# B&R Automation Studio project TD52 (part 4)

#### UniAna_in.st - Implementation file
```iecst
(********************************************************************
 * COPYRIGHT -- INNIO Company, Zengerer
 ********************************************************************
 * Library: AnalogIn
 * File: AnalogIn.st
 * Author: ZengereS
 * Created: December 04, 2007
 ********************************************************************
 *
 * Description of library AnalogIn:
 ********************************************************************
 *  Function depending on ucInputType:
 *  ---------------------------------
 * 		 0=AI_NO_SCALING: 		(Temperature) Inputs  NO SCALING, NO CLAMPING (PT100 or Thermocouples on ATxx- Units, read in 1/10°C)
 *
 * 	THESE INPUT TYPES ARE CLAMPED: (ssScalMin < ssOut < ssScalMax)
 * 		 1=AI_FixedFactor10:	Temperature inputs (PT100, KTY..... WITH FIXED x10 SCALING TO 1°C; CLAMPED
 *		 2=AI_MA_INPUT:			+-20mA input (-32768 to 32767Digits) scaled to ScalMin-ScalMax; CLAMPED
 *		 3=AI_0-20MA_INPUT:		0-20mA input (0-32767Digits) scaled to ScalMin-ScalMax; CLAMPED
 *		 4=AI_4_20MA_INPUT:		4-20mA input (6554-32767Digits) scaled to ScalMin-ScalMax; CLAMPED
  *		 5=AI_0_5V_INPUT:		0-5V input (0-16364Digits) scaled to ScalMin-ScalMax; CLAMPED		(NEW)
 * 		 9=AI_NO_SCALING, CLAMPED: (Temperature) Inputs  NO SCALING (PT100 or Thermocouples on ATxx- Units, read in 1/10°C) ; CLAMPED BETWEEN ScalMin and ScalMax
 *
 *	THESE INPUT TYPES ARE ALLSO AVAILABLE WITHOUT CLAMPING: (ssScalMin <> ssOut <> ssScalMax)
 * 		11=AI_FixedFactor10:	NO CLAMPING Temperature inputs (PT100, KTY..... WITH FIXED x10 SCALING TO 1°C (usage not recommendet)
 *		12=AI_MA_INPUT:			NO CLAMPING +-20mA input (-32768 to 32767Digits) scaled to ScalMin-ScalMax    (usage not recommendet))
 *		13=AI_0-20MA_INPUT:		NO CLAMPING 0-20mA input (0-32767Digits) scaled to ScalMin-ScalMax
 *		14=AI_4_20MA_INPUT:		NO CLAMPING 4-20mA input (6554-32767Digits) scaled to ScalMin-ScalMax
 *		15=AI_0_5V_INPUT:		0-5V input (0-16364Digits) scaled to ScalMin-ScalMax
 *
 *	!scNrOfDecimal WORKS AS MULTIPLIER FOR THE SCALED VALUE BY SHIFTING THE DECIMAL POINT!
 *
 *	DEFINE OUTPUT CHANNELS WITH THESE TYPE CODES: (same sScalMin and ssScalMax are applied to Output signal) (NEESDS EXTERNAL CODE PARTS!)
 * 		11=AI_0-20MA_INPUT:		0-20mA output (0-32767Digits) scaled from channel signal ScalMin-ScalMax (input behavior typ 0, if HW input stays connected!)
 *		24=AI_4_20MA_OUTPUT:	4-20mA output (6554-32767Digits) scaled from channel signal ScalMin-ScalMax (input behavior typ 0, if HW in connected!)
 *
 *
 *  SPECIAL CODES FOR 'usANDLinkNum' (Numbers 1 to 250 are reserved for the channel numbers to add another channel value)
 *		 253=RawManualValue:		Enter MANUAL RAW VALUE in ssManualValue for overriding input
 *		 254=AddManualValue:		Enter MANUAL ADD VALUE in ssManualValue as addition summand to the scaled output
 *		 255=UseManualValue:		Enter MANUAL OVERRIDE VALUE in ssManualValue for direct output
 *
 *	Limit activation with ucOtionBits:
 *  	bErrOptiMin	:= activation with ucOptionBits = 1
 *		bErrOptiMax := activation with ucOptionBits = 2
 *		bErrMin		:= activation with ucOptionBits = 4
 *		bErrMax		:= activation with ucOptionBits = 8
 *		bErrMINMIN	:= activation with ucOptionBits = 16
 *		bErrMAXMAX	:= activation with ucOptionBits = 32

 *  	bErrSignal	:= DEactivation with ucOptionBits = 64   (MEASUREMENT SIGNAL DETECTION-> ALARM)
 *
 ********************************************************************
 *  History:
 *  --------
 *	2008-09-10  V0.20	Zengerer	added scaling calculations
 *	2008-09-11  V0.21	Zengerer	added Helper Structure for old SG3- visu
 *	2008-09-30  V0.22	Zengerer	added texts and color changing
 *	2008-09-30  V0.23	Zengerer	added Input Types 10-14 for unclamped values wihout limitation between Min/Max scaling
 *	2008-10-22  V0.30	Zengerer	CHANGED CONFIGTYPE: scNrOfDecimal instead of ucNrOfDecimal
 *	2009-05-22	V0.40	Zengerer	Limit activation with OtionBits masking
 *	2009-06-22	V0.42	Zengerer	Limit OptionBits update
 *  2010-06-04  V0.50	Zengerer	NAMETEXT expanded to 32 CHARACTERS; ssManualValue and usANDLinkNum new introduced in datatype
  *	2009-11-25	V0.50	Zengerer	0-5V Inputtype added
 *	2010-06-22	V0.51	Zengerer	predefined system value in 'usANDLinkNum' removed here, externaly realised
 *	2010-06-22	V0.52	Zengerer	additional infotext for output types (output handling externaly realised)
 *	2010-06-22	V0.60	Zengerer	Manual override of RAW value! with linkCode 253
 *	2013-10-31	V0.70	Zengerer	FILTER type as local implemented function to cancel dependency on JEW_LIB1
 *  2013-11-11  V0.71	Zengerer	Filter function reverted-  has to stay in task
*
* LEGACY CODE- DO NOT USE IN NEW IMPLEMENTATIONS!
*
 ********************************************************************)

FUNCTION_BLOCK ana_in		(*Analogeingang oder Temperatureingang*)

	IF tAnaInPERMEM.bEnable THEN					(*1=enable input*)
		(*get InputType from parameterstructure: types 1-9 are clamped to min/max EU, types 11-19 are proceedet like 1-9, but without clamping*)
		IF tAnaInPERMEM.ucInputType >9 AND tAnaInPERMEM.ucInputType <19 THEN
			ucInputType	:= tAnaInPERMEM.ucInputType -10;					(*Internal use: input type only from 0-8*)
		ELSE
			ucInputType	:= tAnaInPERMEM.ucInputType ;						(*Internal use: input type only from 0-8*)
			IF tAnaInPERMEM.ucInputType = 9 THEN ucInputType := 0; END_IF	(*Internal use: input type only from 0-8*)
		END_IF

		(*Statustext output*)
		CASE ucInputType OF
			0:		(*AI_NO_SCALING '1234567890123456'*)
					szOutState	:= 	'UnscaledIn(Temp)';
	 		1:		(*AI_AI_FixedFactor10     *)
					szOutState	:= 	'Temp.Input X°C';
			2:		(*AI_-10+10V_INPUT*)
					szOutState	:= 	'+-10V Input OK';
			3:		(*AI_0-20MA_INPUT*)
					szOutState	:= 	'0-20mA OK';
			4:		(*AI_4_20MA_INPUT*)
					szOutState	:= 	'4-20mA OK';
			5:		(*AI_0_5V_INPUT*)
					szOutState	:= 	'+5V Input';
			9:		(*AI_NO_SCALING '1234567890123456'*)
					szOutState	:= 	'Unscaled Clamped';
	 		11:		(*AI_AI_FixedFactor10     *)
					szOutState	:= 	'Temp.Inp.NoClamp';
			12:		(*AI_-10+10V_INPUT*)
					szOutState	:= 	'+-10V In.NoClamp';
			13:		(*AI_0-20MA_INPUT*)
					szOutState	:= 	'0-20mA NoClamp';
			14:		(*AI_4_20MA_INPUT*)
					szOutState	:= 	'4-20mA NoClamp';
			15:		(*AI_0_5V_INPUT*)
					szOutState	:= 	'+5V Inp. NoClamp';
			23:		(*AI_0-20MA_OUTPUT*)
					szOutState	:= 	'0-20mA OUTPUT OK';
			24:		(*AI_4-20MA_OUTPUT*)
					szOutState	:= 	'4-20mA OUTPUT OK';
		ELSE		(*CASE_ELSE*)
					szOutState	:= 	'NoTypeInfo';
		END_CASE

		(*Manual override of RAW value! with linkCode 253 (watch external code allso!*)
		IF tAnaInPERMEM.usANDLinkNum =253 THEN
			ssIn := tAnaInPERMEM.ssManualValue;
		 	szOutState	:= 	'MANUAL RAW VALUE';
		END_IF

		(*SIGNAL FAILURE DETECTION*)
		CASE ucInputType OF
			0:		(*AI_NO_SCALING:  (Temperature inputs PT100, Termocouples == 1/10°C from ATxx Units WITHOUT SCALING *)
				tAna_inErrors.bErrSignal := (ssIn < LIM_PT100_MIN OR ssIn > LIM_PT100_MAX);
			1:		(*AI_AI_FixedFactor10:  (temperature) inputs WITH x10 SCALING to convert to 1°C*)
				tAna_inErrors.bErrSignal := ((ssIn/10) < LIM_PT100_MIN OR (ssIn/10) > LIM_PT100_MAX);
		    2:		(*AI_-10+10V_INPUT*)
				tAna_inErrors.bErrSignal := FALSE;   (*NO SIGNAL CHECK!*)  (* (ssIn < LIM_MA_MIN) *OR ssIn > LIM_MA_MAX); *)
			3:		(*AI_0_20MA_INPUT*)
				tAna_inErrors.bErrSignal := (ssIn < LIM_0_20MA_MIN); (*OR ssIn > LIM_0_20MA_MAX);*)
			4:		(*AI_4_20MA_INPUT*)
				tAna_inErrors.bErrSignal := (ssIn < LIM_4_20MA_MIN); (*OR ssIn > LIM_4_20MA_MAX);*)
			5:		(*AI_0_5V_INPUT*)
				tAna_inErrors.bErrSignal := (ssIn < LIM_0_5V_MIN OR ssIn > LIM_0_5V_MAX);
			9:		(*AI_NO_SCALING, clamped*)
				tAna_inErrors.bErrSignal := (ssIn < LIM_PT100_MIN OR ssIn > LIM_PT100_MAX);
		ELSE		(*CASE_ELSE*)
				tAna_inErrors.bErrSignal := FALSE;

		END_CASE

		(*INPUT SIGNAL FILTER*)
		FILTER_0(In := ssIn, Filter := UINT_TO_USINT(tAnaInPERMEM.usSetFilterValue) );			(*FILTER type local implementedr function to cancel dependency on JEW_LIB1 *)

		IF tAna_inErrors.bErrSignal  THEN
			ssInFiltered := DINT_TO_INT(FILTER_0.Out);
		ELSE
			ssInFiltered := ssIn;		(*unfiltered, to shorten reaction time on signal newstart *)
		END_IF

		(*INPUT SCALING*)
		CASE ucInputType OF
			0:		(*AI_PT100_NO_SCALING*)
					slOutScaled		:= 	INT_TO_DINT( ssInFiltered );
	 		1:		(*AI_AI_FixedFactor10*)
					slOutScaled		:= 	INT_TO_DINT( ssInFiltered ) / 10 ;
			2:		(*AI_-10+10V_INPUT*)
					slOutScaled		:=  (INT_TO_DINT(ssInFiltered) + 32768 ) * (tAnaInPERMEM.ssScalMax - tAnaInPERMEM.ssScalMin) / (32767*2) + tAnaInPERMEM.ssScalMin ;
			3:		(*AI_0-20MA_INPUT*)
					slOutScaled		:= 	(INT_TO_DINT(ssInFiltered)         ) * (tAnaInPERMEM.ssScalMax - tAnaInPERMEM.ssScalMin) / 32768 + tAnaInPERMEM.ssScalMin ;
			4:		(*AI_4_20MA_INPUT*)
					slOutScaled		:=  (INT_TO_DINT(ssInFiltered) - 6554  ) * (tAnaInPERMEM.ssScalMax - tAnaInPERMEM.ssScalMin) / (32768-6554) + tAnaInPERMEM.ssScalMin ;
			5:		(*AI_0_5V_INPUT*)
					slOutScaled		:= 	(INT_TO_DINT(ssInFiltered)         ) * (tAnaInPERMEM.ssScalMax - tAnaInPERMEM.ssScalMin) / 16383 + tAnaInPERMEM.ssScalMin ;			(*scaling 100% = only 50% of electrical max+ to use a +-10V input*)
			9:		(*AI_PT100_NO_SCALING, clamped*)
					slOutScaled		:= 	INT_TO_DINT( ssInFiltered );
		ELSE		(*CASE_ELSE*)
					slOutScaled		:= 	0;
		END_CASE

		(*INPUT CLAMPING on Min-Max scaling parameters*)
		IF tAnaInPERMEM.ucInputType > 0 AND tAnaInPERMEM.ucInputType < 10 THEN	(*all input types with codenumber 1-9 get their output values clamped*)
			IF slOutScaled < tAnaInPERMEM.ssScalMin	THEN slOutScaled := tAnaInPERMEM.ssScalMin;	END_IF
			IF slOutScaled > tAnaInPERMEM.ssScalMax	THEN slOutScaled := tAnaInPERMEM.ssScalMax;	END_IF
		END_IF

		(*OPTION: Calculate combined value of this and another channel*)
		IF tAnaInPERMEM.usANDLinkNum > 0 AND tAnaInPERMEM.usANDLinkNum < 251 THEN
  			(*tAnaInPERMEM.usANDLinkNum; *)  					  	(*!!!	EXTERN realisiert   !!!*)
		 	szOutState	:= 	'Channel x Val.ad';
		END_IF

		(*Add manual value optional with linkCode 254 *)
		IF tAnaInPERMEM.usANDLinkNum =254 THEN
			slOutScaled := slOutScaled + tAnaInPERMEM.ssManualValue;
		 	szOutState	:= 	'Manualvalue add.';
		END_IF
		(*Manual override! with linkCode 255*)
		IF tAnaInPERMEM.usANDLinkNum =255 THEN
			slOutScaled := tAnaInPERMEM.ssManualValue;
		 	szOutState	:= 	'Manual Override';
		END_IF

		(*INPUT CLAMPING ONCE MORE FOR ADDED VALUES*)
		IF tAnaInPERMEM.ucInputType > 0 AND tAnaInPERMEM.ucInputType < 10 THEN	(*all input types with codenumber 1-9 get their output values clamped*)
			IF slOutScaled < tAnaInPERMEM.ssScalMin	THEN slOutScaled := tAnaInPERMEM.ssScalMin;	END_IF
			IF slOutScaled > tAnaInPERMEM.ssScalMax	THEN slOutScaled := tAnaInPERMEM.ssScalMax;	END_IF
		END_IF

		(*OUTPUT TO INTEGER Variable*)
		ssOut 	:= DINT_TO_INT( slOutScaled );
		IF slOutScaled < -32768		THEN ssOut := -32768;	END_IF		(* (just to be sure...) *)
		IF slOutScaled > 32767		THEN ssOut := 32767; 	END_IF   	(* (just to be sure...) *)

		(*		ssOutMod 	:= MOD(ssInFiltered,10);   ALT *)

		(*LIMITS*)
		(*Limit activation with OtionBits masking:  NOT AND=0 (XOR) *)
			tAna_inErrors.bErrOptiMin	:= 	(NOT( (tAnaInPERMEM.ucOptionBits AND 1) =0) ) 		AND (ssOut < tAnaInPERMEM.ssSetPointOptiMin);
  			tAna_inErrors.bErrMin		:= 	(NOT( (tAnaInPERMEM.ucOptionBits AND 4) =0) )		AND (ssOut < tAnaInPERMEM.ssSetPointMin);
  			tAna_inErrors.bErrMINMIN	:= 	(NOT( (tAnaInPERMEM.ucOptionBits AND 16)=0) )		AND (ssOut < tAnaInPERMEM.ssSetPointMINMIN);
			tAna_inErrors.bErrOptiMax	:= 	(NOT( (tAnaInPERMEM.ucOptionBits AND 2) =0) )		AND (ssOut > tAnaInPERMEM.ssSetPointOptiMax);
			tAna_inErrors.bErrMax		:= 	(NOT( (tAnaInPERMEM.ucOptionBits AND 8) =0) )		AND (ssOut > tAnaInPERMEM.ssSetPointMax);
			tAna_inErrors.bErrMAXMAX	:= 	(NOT( (tAnaInPERMEM.ucOptionBits AND 32)=0) )		AND (ssOut > tAnaInPERMEM.ssSetPointMAXMAX);

			(*Statustext Messages for Limits    				'12345678901234'   *)
			IF tAna_inErrors.bErrOptiMin		THEN szOutState	:= 	'<OptiMin exc. '; 	END_IF
			IF tAna_inErrors.bErrMin 			THEN szOutState	:= 	'<Min Limit    '; 	END_IF
			IF tAna_inErrors.bErrMINMIN 		THEN szOutState	:= 	'<MINMIN Limit!'; 	END_IF
			IF tAna_inErrors.bErrOptiMax		THEN szOutState	:= 	'>OptiMax exc. '; 	END_IF
			IF tAna_inErrors.bErrMax 			THEN szOutState	:= 	'>Max Limit    '; 	END_IF
			IF tAna_inErrors.bErrMAXMAX 		THEN szOutState	:= 	'>MAXMAX Limit!'; 	END_IF

		(*Check limit values valid?*)
		(*	IF 	tAnaInPERMEM.bOptSupervice AND*)
   			IF	(NOT( (tAnaInPERMEM.ucOptionBits AND 8)=1 ))	AND			(*Optionsbit für ErrMINMIN ausmaskieren*)
				(NOT( (tAnaInPERMEM.ucOptionBits AND 64)=1 ))	AND			(*Optionsbit für ErrMAXMAX ausmaskieren*)
   				(tAnaInPERMEM.ssSetPointMINMIN = 0) AND
   				(tAnaInPERMEM.ssSetPointMAXMAX <= tAnaInPERMEM.ssSetPointMINMIN)
			THEN
				tAna_inErrors.bErrMINMIN	:= FALSE;
				tAna_inErrors.bErrMAXMAX	:= FALSE;
				szOutState	:= 	'LimitsNotValid';
			END_IF

		IF tAna_inErrors.bErrSignal  THEN	szOutState	:= 	'OutOfRange'; END_IF

		(*failed signal check sets output to 'errorvalue' *)
		IF tAna_inErrors.bErrSignal AND NOT (tAnaInPERMEM.usANDLinkNum =255) THEN
			ssOut		:= -9999;
(*			ssOutModulo	:= -9999; 	*)
		END_IF
		IF tAnaInPERMEM.usANDLinkNum =255 THEN	szOutState	:= 	'Manual Override!'; 	END_IF 	(*this messagetext has priotity and overrides the one before!*)

		(*Quittierung...*)
			bInQuit;
		(* 	bOutErr		:= FALSE;
		(*FEHLT NOCH!!!*)

		(*Config Mode*)
		(*FEHLT NOCH!!!*)
		(*bConfigModeActive;*)

	ELSE						(* else to .bEnable: 0=disables all input functions*)
		ssOut		:= 0;
		ssOutModulo	:= 0;
		rOut		:= 0;
		tAna_inErrors.bErrSignal 	:= 	FALSE;
		tAna_inErrors.bErrMAXMAX	:= 	FALSE;
		tAna_inErrors.bErrMax		:= 	FALSE;
		tAna_inErrors.bErrOptiMax	:= 	FALSE;
		tAna_inErrors.bErrOptiMin	:= 	FALSE;
		tAna_inErrors.bErrMin		:= 	FALSE;
		tAna_inErrors.bErrMINMIN	:= 	FALSE;
		szOutState	:= 	'DISABELED';

	END_IF

	(*Alternative: output as scaled real value*)
(*OLD	CASE tAnaInPERMEM.scNrOfDecimal  OF
			-1:		(**)
(*					rOut			:= INT_TO_REAL(ssOutScaled) *10 ;
			0:
(*					rOut			:= INT_TO_REAL(ssOutScaled);
			1:		(**)
(*					rOut			:= INT_TO_REAL(ssOutScaled) /10 ;
			2:		(**)
(*					rOut			:= INT_TO_REAL(ssOutScaled) /100 ;
			3:		(**)
(*					rOut			:= INT_TO_REAL(ssOutScaled) /1000 ;
			4:		(**)
(*					rOut			:= INT_TO_REAL(ssOutScaled) /10000 ;
	ELSE		(*CASE_ELSE*)
(*					rOut			:= 0 ;
	END_CASE		(**)

		rOut		:= DINT_TO_REAL(slOutScaled)  * EXPT(10 , -tAnaInPERMEM.scNrOfDecimal) ;  (* ...*10^(-NrOfDecimal) VORSICHT: NICHT IEC1131 -Konform!!*)

END_FUNCTION_BLOCK

(******************************************************************************)
(******************************************************************************)
(******************************************************************************)

FUNCTION_BLOCK ana_in_SG3helper		(*stellt mit Informationen aus ana_in zusäzlichen Statusausgängen für alte SG3- Visu zur Verfügung*)

		(*outputs for local paneldisplay*)
(*OLD*		CASE ucInputType OF
(*	 		0:		(*AI_NO_SCALING*)
(*					ssOutRaw		:= 	DINT_TO_INT( LIMIT( (INT_TO_DINT(ssInRaw)   * 32767  / 2000 )    , 0, 32767) ); (*scale 0-200°C to full display range*)
(*			1:		(*AI_PT100_NO_SCALING*)
(*					ssOutRaw		:= 	DINT_TO_INT( LIMIT( (INT_TO_DINT(ssInRaw)   * 32767  / 2000 )    , 0, 32767) ); (*scale 0-200°C to full display range*)
(*			2:		(*AI_-10+10V_INPUT*)
(*					ssOutRaw		:= 	LIMIT( ABS( ssInRaw )  	, 0, 32767);
(*			3:		(*AI_0-20MA_INPUT*)
(*					ssOutRaw		:= 	LIMIT( ssInRaw  		, 0, 32767);
(*			4:		(*AI_4_20MA_INPUT*)
(*					ssOutRaw		:= 	LIMIT( ssInRaw  		, 0, 32767);
(*		ELSE
(*					ssOutRaw		:= 	LIMIT( ssInRaw  		, 0, 32767);
(*		END_CASE
(*\OLD*)
	(*	ssOutRaw		:= 	REAL_TO_INT( LOG( INT_TO_REAL(ssInRaw) / 100 ) * 13000 );		(*logarythmic bargraph scaling*)
	(*	ssOutRaw		:= 	REAL_TO_INT( LN( INT_TO_REAL(ssInRaw) ) * 3150 );		(*logarythmic bargraph scaling*)
		ssOutRaw		:= 	REAL_TO_INT( SQRT( INT_TO_REAL(ssInRaw) ) * 181 );		(*exponential bargraph scaling*)

		(*OPTIONAL: outputs scaled for local paneldisplay with fixed 3 digits after decimal*)
		CASE tAnaInPERMEM.scNrOfDecimal  OF
	 		0:
					slOut			:= DINT_TO_INT(ssIn) * 1000;
			1:		(**)
					slOut			:= DINT_TO_INT(ssIn) * 100 ;
			2:		(**)
					slOut			:= DINT_TO_INT(ssIn) * 10;
			3:		(**)
					slOut			:= DINT_TO_INT(ssIn) * 1;
			4:		(**)
					slOut			:= DINT_TO_INT(ssIn) / 10;

		ELSE		(*CASE_ELSE*)
					slOut			:= 0 ;
		END_CASE

	(*SG3 VISU: HELPER OUTPUTS to activate displays and change colors*)
 	tAnaInHelper.ucStatus	:= 93;														(* blue and INvisible (set 1-bit == uneven decimal colornumber)*)
	IF  tAnaInPERMEM.bEnable	 THEN
 		tAnaInHelper.ucStatus	:= 10;													(* green and visible (no 1-bit! == only even decimal numbers)*)
		IF 	tAna_inErrors.bErrOptiMax OR tAna_inErrors.bErrOptiMin	THEN  	tAnaInHelper.ucStatus := 142; END_IF	(* (ligth)green and visible (no 1-bit!*)
		IF 	tAna_inErrors.bErrMax OR tAna_inErrors.bErrMin			THEN  	tAnaInHelper.ucStatus := 040; END_IF	(* yellow and visible (no 1-bit!*)
		IF 	tAna_inErrors.bErrMAXMAX OR tAna_inErrors.bErrMINMIN	THEN  	tAnaInHelper.ucStatus := 050; END_IF	(* red and visible (no 1-bit!*)
  		IF 	tAna_inErrors.bErrSignal								THEN  	tAnaInHelper.ucStatus := 038; END_IF	(* red and visible (no 1-bit!*)
		IF ssInRaw < - 4											THEN	tAnaInHelper.ucStatus := 246; END_IF	(* NEGATIVE RAW VALUES showed liggthblue and visible (no 1-bit!*)

	(*SG3 VISU: HELPER OUTPUTS to activate displays with different No of digits after decimal point*)
		CASE tAnaInPERMEM.scNrOfDecimal OF
	 		0:
					tAnaInHelper.ucStatus0Digits := 0;
					tAnaInHelper.ucStatus1Digits := 1;
					tAnaInHelper.ucStatus2Digits := 1;
					tAnaInHelper.ucStatus3Digits := 1;
					tAnaInHelper.ucStatus4Digits := 1;
	 		1:
					tAnaInHelper.ucStatus0Digits := 1;
					tAnaInHelper.ucStatus1Digits := 0;
					tAnaInHelper.ucStatus2Digits := 1;
					tAnaInHelper.ucStatus3Digits := 1;
					tAnaInHelper.ucStatus4Digits := 1;
	 		2:
					tAnaInHelper.ucStatus0Digits := 1;
					tAnaInHelper.ucStatus1Digits := 1;
					tAnaInHelper.ucStatus2Digits := 0;
					tAnaInHelper.ucStatus3Digits := 1;
					tAnaInHelper.ucStatus4Digits := 1;
	 		3:
					tAnaInHelper.ucStatus0Digits := 1;
					tAnaInHelper.ucStatus1Digits := 1;
					tAnaInHelper.ucStatus2Digits := 1;
					tAnaInHelper.ucStatus3Digits := 0;
					tAnaInHelper.ucStatus4Digits := 1;
	 		4:
					tAnaInHelper.ucStatus0Digits := 1;
					tAnaInHelper.ucStatus1Digits := 1;
					tAnaInHelper.ucStatus2Digits := 1;
					tAnaInHelper.ucStatus3Digits := 1;
					tAnaInHelper.ucStatus4Digits := 0;
		END_CASE

	ELSE	(*hide displays...*)
 			tAnaInHelper.ucStatus	:= 1;

			tAnaInHelper.ucStatus0Digits := 1;
			tAnaInHelper.ucStatus1Digits := 1;
			tAnaInHelper.ucStatus2Digits := 1;
			tAnaInHelper.ucStatus3Digits := 1;
			tAnaInHelper.ucStatus4Digits := 1;
	END_IF

END_FUNCTION_BLOCK
```

#### UniAna_in.typ - Exported data types
```iecst
(********************************************************************
 * COPYRIGHT -- INNIO Company, Zengerer
 ********************************************************************
 * Library: AnalogIn
 * File: AnalogIn.typ
 * Author: ZengereS
 * Created: December 04, 2007
*  V1.1 2010-06-20
 ********************************************************************
 * Data types of library AnalogIn
 ********************************************************************)

TYPE
	tAnaInPERMEM_typ : 	STRUCT
		bEnable : BOOL; (*0 disables input function and all depending alarms*)
		ucInputType : USINT; (*can be set or will be default: temp. x10 °C, if not used*)
		ssScalMin : INT; (*min. engineering units at lower end of input range; not necessary for temp.*)
		ssScalMax : INT; (*min. engineering units at lower end of input range; not necessary for temp.*)
		usSetFilterValue : UINT; (*Optional signal filtering: 0=no Filter, 64000=max. input damping*)
		bOptSupervice : BOOL; (*Set to 1, if SIGNAL ERROR or MINMIN or MAXMAX will trigger ALARM (PRIO3)*)
		ssSetPointMAXMAX : INT; (*Optional limit value (for warning+ possible alarm shutdown)*)
		ssSetPointMax : INT; (*Optional limit value (for warning message)*)
		ssSetPointOptiMax : INT; (*Optional limit value*)
		ssSetPointOpti : INT; (*Optional limit value*)
		ssSetPointOptiMin : INT; (*Optional limit value*)
		ssSetPointMin : INT; (*Optional limit value (for warning message)*)
		ssSetPointMINMIN : INT; (*Optional limit value (for warning+ possible alarm shutdown)*)
		tiSetMaxMaxTime : TIME; (*Optional Delay time for Max and MAXMAX Alarms*)
		tiSetMinMinTime : TIME; (*Optional Delay time for Min and MINMIN Alarms*)
		scNrOfDecimal : SINT; (*No of digits after decimal point on display or real output*)
		szHardware : STRING[16]; (*Optional Text for Visualisation*)
		szChannelName : STRING[32]; (*Optional Text for Visualisation*)
		szUnit : STRING[6]; (*Optional Text for Visualisation*)
		ucOptionBits : USINT; (*Message enabling bitfield: 0=all imit messages are disabeled*)
		ssManualValue : INT; (*Optional used Value for manual override(255) or add to channelvalue (254)...*)
		usANDLinkNum : UINT; (*Cannel Number to add value (or 255 for manual override)*)
	END_STRUCT;
	tAnaInHelper_typ : 	STRUCT
		ucStatus : USINT; (*outputs 0,if input is enabled and 1 to hide disabled inputs*)
		ucStatus0Digits : USINT; (*outputs 0, if no digit after decimal point is selected*)
		ucStatus1Digits : USINT; (*outputs 0, if 1 digit after decimal point is selected*)
		ucStatus2Digits : USINT; (*outputs 0, if 2 digits after decimal point is selected*)
		ucStatus3Digits : USINT; (*outputs 0, if 3 digit after decimal point is selected*)
		ucStatus4Digits : USINT; (*outputs 0, if 4 digit after decimal point is selected*)
	END_STRUCT;
	tAnaInErrors_typ : 	STRUCT
		bErrMAXMAX : BOOL; (*status: value is above MaxMax level*)
		bErrOptiMax : BOOL; (*status: value is above OptiMax level*)
		bErrMax : BOOL; (*status: value is above Max level*)
		bErrOptiMin : BOOL; (*status: value is below OptiMin level*)
		bErrMin : BOOL; (*status: value is below Min level*)
		bErrMINMIN : BOOL; (*status: value is below MinMin level*)
		bErrSignal : BOOL; (*digital error output (Signal Error or MAXMAX/MINMIN exceedet)*)
	END_STRUCT;
END_TYPE
```

#### UniAna_in.var - Exported constants
```iecst
(********************************************************************
 * COPYRIGHT -- INNIO Company
 ********************************************************************
 * Library: AnalogIn
 * File: AnalogIn.var
 * Author: ZengereS
 * Created: December 04, 2007
 ********************************************************************
 * Constants of library AnalogIn
 ********************************************************************)
VAR CONSTANT
	tiDefaultAlarmDelayTime : TIME := T#5s; (*Vorgabewert Verzögerung bis Alarm (vor Programmierung)*)
	AI_PT100_NO_SCALING : USINT := 1; (*temperature value, scaling x10*)
	AI_NO_SCALING : USINT := 0; (*+-value, scaling setpoints are not used*)
	AI_V_INPUT : USINT := 2; (*Analog Input, scaled from -10V to +10V =-32767 to 32767*)
	AI_0_20MA_INPUT : USINT := 3; (*Analog Input, scaled from 0-20mA  =0 to 32767*)
	AI_4_20MA_INPUT : USINT := 4; (*Analog Input, scaled from 4-20mA =6540 to 32767*)
	LIM_PT100_MIN : INT := -1990; (*signal error limit value for -199°C*)
	LIM_PT100_MAX : INT := 32000; (*signal error limit value for 3200°C*)
	LIM_MA_MIN : INT := -32768; (*signal error limit value for -20mA*)
	LIM_0_20MA_MIN : INT := -1638; (*signal error limit value for -1mA*)
	LIM_4_20MA_MIN : INT := 4915; (*signal error limit value for 3mA*)
	LIM_0_5V_MIN : INT := -3276; (*signal error limit value for -1V*)
	LIM_0_5V_MAX : INT := 19660; (*signal error limit value for +6V*)
END_VAR
```

#### UniAna_in.fun - Exported functions and function blocks
```iecst
(********************************************************************
 * COPYRIGHT -- INNIO Company
 ********************************************************************
 * Library: AnalogIn
 * File: AnalogIn.fun
 * Author: ZengereS
 * Created: December 04, 2007
 ********************************************************************
 * Functions and function blocks of library AnalogIn
 ********************************************************************)

FUNCTION_BLOCK ana_in
	VAR_INPUT
		ssIn : INT; (*Analog input from hardware*)
		bInQuit : BOOL; (*quitt error messages input*)
		tAnaInPERMEM : tAnaInPERMEM_typ; (*Assign Variable to Permanent Memory!*)
	END_VAR
	VAR_OUTPUT
		ssOut : INT; (*compatible OLD integer scaled analoge value*)
		ssOutModulo : INT; (*modulo of scaled value, if >0 digits after . selected in parameter*)
		rOut : REAL; (*altenative output as scaled real value*)
		szOutState : STRING[16]; (*status output in clear text for visualisation*)
		tAna_inErrors : tAnaInErrors_typ; (*statusbits for error indication*)
	END_VAR
	VAR
		slOutScaled : DINT; (*Do Not Use- Internal use only*)
		ssInFiltered : INT; (*Do Not Use- Internal use only*)
		ucInputType : USINT; (*Do Not Use- Internal use only*)
		FILTER_0 : xUniAnaFilter;
	END_VAR
END_FUNCTION_BLOCK

FUNCTION_BLOCK ana_in_SG3helper
	VAR_INPUT
		ssInRaw : INT; (*Analog input from hardware*)
		ssIn : INT; (*OPTIONAL: scaled analog input from output of scaling function*)
		tAna_inErrors : tAnaInErrors_typ; (*statusbits for error indication*)
		tAnaInPERMEM : tAnaInPERMEM_typ; (*Assign Variable to Permanent Memory!*)
	END_VAR
	VAR_OUTPUT
		ssOutRaw : INT; (*scaled analoge value,*)
		slOut : DINT; (*OPTIONAL: scaled analoge value FOR FIXED 3DIGITS AFTER DECIMAL DISPLAY*)
		tAnaInHelper : tAnaInHelper_typ; (*helper bits data type, especialy for older SG3- visualisation*)
	END_VAR
END_FUNCTION_BLOCK

FUNCTION_BLOCK xUniAnaFilter (* filter with PT1 behaivior and DINT in/output *)
	VAR_INPUT
		In : DINT;
		Filter : UINT;
	END_VAR
	VAR_OUTPUT
		Out : DINT;
	END_VAR
	VAR
		mw : DINT;
	END_VAR
END_FUNCTION_BLOCK

FUNCTION_BLOCK xUniAnaFilterR (* filter with PT1 behaivior and REAL in/output *)
	VAR_INPUT
		In : REAL;
		Filter : UINT;
	END_VAR
	VAR_OUTPUT
		Out : REAL;
	END_VAR
	VAR
		mw : REAL;
	END_VAR
END_FUNCTION_BLOCK
```

#### UniAnaFilter.st
```iecst
(********************************************************************
 * COPYRIGHT -- Bernecker + Rainer
 ********************************************************************
 * Package: UniAna_in
 * File: UniAnaFilter.st
 * Author: froehlichw
 * Created: November 30, 2011
 ********************************************************************
 * Implementation COPIED FROM THE function block HALioFilter
 *
 * History:
 * 14.12.2011  V0.00.0 froehlichw
 *      (new)  created
 *******************************************************************)

FUNCTION_BLOCK xUniAnaFilter

	(* avoid division by 0 *)
	IF (Filter = 0) THEN
		Filter:= 1;
	END_IF;
	mw:= mw + In - Out;
	Out:= mw/UINT_TO_DINT(Filter);

END_FUNCTION_BLOCK
```

#### UniAnaFilterR.st
```iecst
(********************************************************************
 * COPYRIGHT -- Bernecker + Rainer
 ********************************************************************
 * Package: UniAna_in
 * File: UniAnaFilterR.st
 * Author: froehlichw
 * Created: November 30, 2011
 ********************************************************************
 * Implementation COPIED OF FROM function block HALioFilterR
 *
 * History:
 * 14.12.2011  V0.00.0 froehlichw
 *      (new)  created
 *******************************************************************)

FUNCTION_BLOCK xUniAnaFilterR

	(* avoid division by 0 *)
	IF (Filter = 0) THEN
		Filter:= 1;
	END_IF;
	mw:= mw + In - Out;
	Out:= mw/UINT_TO_REAL(Filter);

END_FUNCTION_BLOCK
```

### Library Logical/Libraries/UniDig_in (IEC, version 0.61.0) - LEGACY CODE- DO NOT USE IN NEW IMPLEMENTATIONS!

#### UniDig_in.typ - Exported data types
```iecst
(********************************************************************
 * COPYRIGHT -- INNIO Company, Zengerer
 ********************************************************************
 * Library: AnalogIn
 * File: AnalogIn.typ
 * Author: ZengereS
 * Created: December 04, 2007
 ********************************************************************
 * Data types of library AnalogIn
 ********************************************************************)

TYPE
	tDigInPERMEM_typ : 	STRUCT
		bEnable : BOOL; (*0 disables channel function and all depending alarms*)
		szChannelName : STRING[32]; (*Optional Text for Visualisation*)
		szHardware : STRING[16]; (*Optional Text for Visualisation (Input or Output Hardwarename)*)
		ucInputType : USINT; (*can be set or will be default: 0=only with visu parameter on/off, 1=OR hardware input, 2=OR ....*)
		bManualOn : BOOL; (*TRUE= set output TRUE (with TON and messages as configured), 0=output depending on ucInputType*)
		bManualBlock : BOOL; (*TRUE= set output FALSE (with TOF and messages as configured), 0= output depending on ucInputType*)
		usORLinkNum : UINT; (*Optional link channel source number for OR- logic*)
		usANDLinkNum : UINT; (*Optional digital link channel source number for AND logic*)
		ulSetTONTime : UDINT; (*Optional TON Delay time*)
		ulSetTOFTime : UDINT; (*Optional TOF Delay time*)
		ucButtonLevel : USINT; (*minimum user level required for button/ channel actions*)
		ucOptionBits : USINT; (*Optional enabling bits: 1=OnWarn, 2=OnAlarm, 4=OffWarn, 8=OffAlarm, 16=CounterLimitWarn*)
		ulCounterLimit : UDINT; (*Optional Eventcounter Limit; !Enable bOptAlarmOn or WarnOn to use!*)
		ulCounter : UDINT; (*Optional Eventcounter Limit; !Enable bOptAlarmOn or WarnOn to use!*)
	END_STRUCT;
	tDigIn_SG3helper_typ : 	STRUCT
		ucStatus : USINT; (*True/ False... State for TextAdvanced*)
		usSetState : USINT; (*True/ False... State for TextAdvanced INPUT*)
		usHideButtonOn : USINT; (*Visibility of Button: 1=hide*)
		usHideButtonOff : USINT; (*Visibility of Button: 1=hide*)
	END_STRUCT;
	tDigInErrors_typ : 	STRUCT
		bErrOnAlarm : BOOL; (*status: value is on*)
		bErrOnWarn : BOOL; (*status: value is above Max level*)
		bErrOffWarn : BOOL; (*status: value is off*)
		bErrOffAlarm : BOOL; (*status: value is below MinMin level*)
		bOnMessage : BOOL;
		bOffMessage : BOOL;
	END_STRUCT;
END_TYPE

(*Insert your comment here.*)
(*Insert your comment here.*)
```

#### UniDig_in.var - Exported constants
```iecst
(********************************************************************
 * COPYRIGHT -- INNIO Company
 ********************************************************************
 * Library: AnalogIn
 * File: AnalogIn.var
 * Author: ZengereS
 * Created: December 04, 2007
 ********************************************************************
 * Constants of library AnalogIn
 ********************************************************************)
VAR CONSTANT
	tiDefaultWarnDelayTime : TIME := T#2s; (*Vorgabewert Verzögerung bis Warning (vor Programmierung)*)
	tiDefaultTONTime : TIME := T#2s; (*Vorgabewert Verzögerung Signal Ein (vor Programmierung)*)
	tiDefaultTOFTime : TIME := T#10ms; (*Vorgabewert Verzögerung Signal Aus (vor Programmierung)*)
END_VAR
```

#### UniDig_in.fun - Exported functions and function blocks
```iecst
(********************************************************************
 * COPYRIGHT -- INNIO Company
 ********************************************************************
 * Library: DiglogIn
 * File: DigIn.fun
 * Author: ZengereS
 * Created: December 20, 2008
 ********************************************************************
 * Functions and function blocks of library DigitalIn
 *******************************************************************
* FUNCTIONS NO LONGER USED! Lib files for declaration only.*)

FUNCTION_BLOCK dig_in
	VAR
		slOutScaled : DINT; (*Do Not Use- Internal use only*)
		ssInFiltered : INT; (*Do Not Use- Internal use only*)
		ucInputType : USINT; (*Do Not Use- Internal use only*)
	END_VAR
END_FUNCTION_BLOCK
```

#### UniDig_in.st - Implementation file
```iecst
(*** OLD! ONLY USED FOR TYPEDECLARATIONS. NO FUNCTIONS USED ANYMORE for digital channels.  ****)

(********************************************************************
 * COPYRIGHT -- INNIO Company, Zengerer
 ********************************************************************
 * Library: DigitalIn
 * File: DigIn.st
 * Author: ZengereS
 * Created: Jan 12, 2009
 ********************************************************************
 *
 * Description of library AnalogIn:
 ********************************************************************
 *  Function depending on ucInputType:
 *  ---------------------------------
 * 	THESE INPUT TYPES ARE AVAILABLE:
 * 		 0=NO_OR_LINK: 					Channel status only set by visu parameter (default)
 * 		 1=OR Hardware Digital IN Nr:	Channel connected to predefined hardware input channel
 *		 2=OR AI_LimitMax Nr:			Channel connected to Analog Input Limit
 *		 4=OR AI_LimitOptiMax Nr:		Channel connected to Analog Input Limit
 *		 8=OR AI_LimitOptiMin Nr:		Channel connected to Analog Input Limit
 * 	   128=OR UniversalDigtal Nr:		Channel connected to reuse other digital channel
 *
 ********************************************************************
 *  History:
 *  --------
 *	2009-02-08  V0.20	Zengerer	1.st type definition
 *	2019-11-13  V0.21	Zengerer	DUMMY LIB without any function; call to avoid compiler warning 5880
 *
 * LEGACY CODE- DO NOT USE IN NEW IMPLEMENTATIONS!
 *
 ********************************************************************)

FUNCTION_BLOCK dig_in		(*Eingang*)
	(* Dummy function, to avoid compiler warning 5880 *)
	slOutScaled ; 	(*Do Not Use- Internal Dummy*)
	ssInFiltered ; 	(*Do Not Use- Internal Dummy*)
	ucInputType ; 	(*Do Not Use- Internal Dummy*)

	(* remove library, when not longer needed for para tape compatibility. *)

END_FUNCTION_BLOCK
```

### Library Logical/Libraries/UniXMLStri (IEC, version 0.44.0) - LEGACY CODE- DO NOT USE IN NEW IMPLEMENTATIONS!

#### UniXMLStri.st
```iecst
	(********************************************************************************************************************
	* Code and Decode XML Data and String composition FOR UNIVERSAL IO Parameter!
	* Copyright 2010 GE Jenbacher
	*
	* History:
	* --------
	* V0.10	12.11.10, Zengerer		generated
	* V0.20	02.12.10, Zengerer		xUniDecoString functin ok with * as wildcard
	* V0.21	16.12.10, Zengerer		unused varname warnings solved
	* V0.30	17.01.11, Zengerer		tUniCalcCheckSumm new
	* V0.40 20.01.11, Zengerer		InMemAdress and InMemLenght as alternative Inputs for tUniCalcCheckSumm
	* V0.41 25.01.11, Ze			szWildcard[1] := '/' (urgent!)
	* V0.42 01.02.11, Ze			No Error Message if characteri s not foun
	* V0.43	04.02.11, Zengerer		Stingdeclarations from 255->300 character
	* V0.44	09.02.11, Zengerer		Errorr message
	*
	* LEGACY CODE- DO NOT USE IN NEW IMPLEMENTATIONS!
	*
	* Description:
	* ------------
	* - xUniDecoXML.fun
	* read parameter from string (XML data line)
	*
	* - xUniCodXML.fun
	* write parameter to string (XML data line)
	*
	* - tUniCalcCheckSumm
	* calculates a alternating checksumm for a string (up to 255chr)
	*
	*
	(* FUNCTION INTERFACE: VALID LIMITATIONS:	*)
	(* --------------------------------------	*)
	(*INPUTS:*)
	(*	bEnable : BOOL; (*TRUE = enable FUB*)
	(*	szConfigString : STRING[255]; (*String holding the data, in wich separatorstrings where searched. Minimum string lenght is the separator string lengt *)
	(*	szSeparator : STRING[10]; (*Enter a combination of detectable separator characters here; wildcard is the * (=position will be ignored)*)
	(*	ucStartPos : USINT; (*position of first character in string to start searching*)

	(*OUTPUTS: *)
	(*	usErrorCode : UINT; (*0=OK or ready without errors, 1=busy, other error numbers see in code*)
	(*	usFoundPos : UINT; (*position of first data character after the found separator*)
	(*	usFoundLenght : UINT; (*lenght of data in characters after the found separator*)
	(*	bLastData : BOOL; (*TRUE, if no more separators will follow afther the found one*)

	(********************************************************************************************************************)
FUNCTION_BLOCK xUniCodString
	(****************************************************************************************************************)
	(* Decode WHOLE PARAMETERSTRUCTURE INFORMATION FROM Textstring
	(****************************************************************************************************************)

	IF bEnable THEN
	//  FEHLT NOCH

	(*	VAR_INPUT*)
		bEnable ;
		ulXMLDataAdress ;
		ulXMLDataSize ;

	(*VAR_OUTPUT *)
		bErrUniXMLRead ;
		usErrorCode ; (*0=OK, ready*)
		bUniAnaFileReadDone ;

	(*VAR*)
		bUniXMLWrite;
		step ;
	END_IF

END_FUNCTION_BLOCK

	(********************************************************************************************************************)
FUNCTION_BLOCK xUniDecoString
	(****************************************************************************************************************)
	(* Decode WHOLE PARAMETERSTRUCTURE INFORMATION FROM Textstring
	(****************************************************************************************************************)

	IF bEnable THEN
		usErrorCode := 1;				(*set state to BUSY*)

		szWildcard[0] := '*' ;
		szWildcard[1] := '/' ;
//old	ucMaxNoOfWildcards := 3;	(*max. allowed number of wildcards to ignore*)

		usFoundPos 		 := 0;
		usFoundLenght	 := 0;
		ucFoundWildcards := 0;
		bLastData		 := FALSE;

		(*examine ConfigString*)
 		usUniStringLen 	:= LEN(szConfigString);
 		usUniSepaLen 	:= LEN(szSeparator);
		IF usUniSepaLen < 2 OR usUniSepaLen > 16 THEN 	(*check for valid separator characters*)
			szSeparator := '|*=';
			usUniSepaLen := 3;
			usErrorCode := 63001;		(*Error: invalid separator string recived*)
		END_IF
  		IF usUniStringLen < usUniSepaLen+1 THEN 		(*minimum string lenght is the lenght of one separator sequenze +1*)
			CNr := usUniStringLen;		(*= exit, no more function *)
			usErrorCode := 63002;		(*Error: empty or to short string recived*)
		END_IF
 		IF usUniStringLen >254 THEN 	(*maximum string lenght*)
			CNr := 255;					(*= exit, no more function *)
			usErrorCode := 63003;		(*Error: to long string recived*)
		END_IF
		IF ucStartPos = 0 THEN
			ucStartPos := 1;
			usErrorCode := 63004;		(*Error: missing startposition entered*)
		END_IF
		IF ucStartPos > usUniStringLen THEN
			CNr := 255;					(*= exit, no more function *)
			usErrorCode := 63005;		(*Error: illegal startposition entered*)
		END_IF

		FOR Sepa := 1 TO usUniSepaLen DO				(*Splitt Separatorstring in single characters*)
			szSepar[Sepa] := MID(szSeparator,1,Sepa);
		END_FOR

		(*detect known separators*)
			CNr := ucStartPos ;											(*start position in string*)

			WHILE CNr <= usUniStringLen DO
				szCNr := MID(szConfigString,1,CNr);						(*get single character at actual position*)

				IF szSepar[1] = szCNr THEN								(*look for 1st separator character*)
					bFound	:= TRUE;									(*start assuming, that this could be a match*)
					ucFoundSlashs := 0;
					CNr		:= CNr + 1;
					CNrStartDetailSearch := CNr;						(*Store startpoint of FollowingCharacterSearch for latrer use in case of missmatch *)
					Sepa 	:= 2;
					(*FEHLT NOCH: restlängenprüfung*)

					(*IF 1ST separator is found, THEN cycle trough following characters*)
					WHILE Sepa < usUniSepaLen+1 DO  						(*check all following separator character*)
						szCNr := MID(szConfigString,1,CNr);					(*get single character at actual position*)

						IF szSepar[Sepa] = szCNr THEN
								Sepa := Sepa +1;							(*A: if matching separator character found, go on to next sepa (and next character) ...*)

						ELSE												(*B: if not, then check, if this separatorposition or this stringposition has a reason to be ignored...*)
							IF szSepar[Sepa] = szWildcard[0]  THEN 			(*	 B1: check, if to ignore wildcard on this separator position *)
								ucFoundWildcards := ucFoundWildcards+1;
								Sepa := Sepa +1;

								IF ucFoundWildcards > 3 THEN		//ucMaxNoOfWildcards THEN
									ucFoundWildcards := 0;
									usErrorCode := 65000 + Sepa;				(*Error: more than max. allowed number of wildcards to ignore*)
									bFound := FALSE;
								END_IF

							ELSE											(*	 B2: if not, check, if ignorable / character is in searchstring *)
								IF szCNr = szWildcard[1]  THEN 				(*ignore / in DATA to recognize XML endtag with same definition as starttag definition *)
									ucFoundSlashs := ucFoundSlashs + 1;

									IF ucFoundSlashs > 2 THEN  		// ucMaxNoOfSlashs THEN
										Sepa := Sepa +1;
										ucFoundSlashs := 0;
										usErrorCode := 65100 + Sepa;			(*Error: more than max. allowed number of slash characters found to ignore*)
										bFound := FALSE;
									END_IF

									CNr ; //:= 	CNr + 1;						(* do not increment here (automatic increment at end of while loop) *)
			//böse!					IF Sepa > 0 THEN Sepa := Sepa -1; END_IF	(*NEVER DO THIS! because of CNr = CNr - Sepa	*)

								ELSE										(*C: if not found, then this character is realy wrong here, so...  *)
									bFound := FALSE; 						(*   ..clear match assumption flag... *)
									CNr		:= CNrStartDetailSearch; //CNr - Sepa;		(*   ..go back in searchstring to the start of detail search...  *)
									Sepa := usUniSepaLen +1;				(*   ..and set exit condition for this while loop.  *)
								//	usErrorCode := 64000+CNr;				(*DO NOT GENERATE ERROR HERE! Error message: wrong character found at pos.*)
									ucFoundWildcards := 0;
								END_IF
							END_IF
						END_IF

						CNr := 	CNr +1;									(*try next character*)
					END_WHILE	(*END INNER CYCLE*)

					IF bFound THEN
						IF usFoundPos = 0 THEN							(*This is the first valid separator*)
	 						usFoundPos := CNr;							(*=FB OUTPUT*)
							usFoundLenght := 0;
							ucFoundWildcards := 0;
							bFound := FALSE;
						ELSE											(*This is the second valid separator*)
	 						usFoundLenght := CNr - usFoundPos - usUniSepaLen ;	(*=FB OUTPUT*)

							ucFoundWildcards := 0;
							bFound := FALSE;
							IF CNr > usUniStringLen THEN				(*End of string reached...*)
   								bLastData := TRUE;
   							END_IF
							CNr := 255;									(*EXIT THE WHILE LOOP and so EXIT FUNCTION, if 2nd valid separatorstring is found *)
						END_IF
					ELSE
						CNr := CNrStartDetailSearch ; //+ 1;				(*retry search for 1st Sepa with next CNr in String*)
					END_IF

				ELSE													(*look for 1st separator character-> NOT FOUND*)
					CNr := 	CNr +1;			(*<-YOU ARE HERE*)			(*try next character*)								(*try next character*)
				END_IF

			END_WHILE			(*END OUTER CYCLE OVER ALL CHARACTERS*)
			IF CNr <> 255 THEN
				IF usFoundPos > 0 THEN
					usFoundLenght := usUniStringLen - usFoundPos + 1;
				END_IF							(*= only 1 valid separator was found, so all the rest of the string is data to this separator *)
												(*Detect End of string reached: if while loop has terminated without rigid setting of CNr := 255.. *)
	   			bLastData := TRUE;
	   		END_IF

  		IF usErrorCode = 1 THEN usErrorCode := 0;  END_IF 	(*set state from BUSY to READY, if no errors occured*)

		(*OLD:	ucFoundSepNr : USINT; ( *Internal*)

	END_IF

END_FUNCTION_BLOCK

	(********************************************************************************************************************)
FUNCTION_BLOCK xUniCalcCheckSumm
	(****************************************************************************************************************)
	(* 	* calculates a alternating checksumm FOR a STRING (up TO 255chr)
	(****************************************************************************************************************)

	IF bEnable THEN
		usErrorCode := 1;				(*set state to BUSY*)
		ssChecksumm	:= 0;
		bPair 			:= FALSE;

		IF InMemAdress > 0 AND InMemLenght > 0 THEN
 			ulADRString		:=  InMemAdress;
			usUniStringLen	:= 	InMemLenght;
		ELSE
			ulADRString		:= ADR(InString);
			usUniStringLen	:= LEN(InString);
		END_IF
		IF usUniStringLen > 1000  THEN
 			usErrorCode := 23456;	(*Checksumm Data array unreliable big*)
		ELSE
			CASE usChecksummMode OF
	  			0:	(*alternating character summ (11er) *)
					FOR CNr := 0 TO usUniStringLen DO
						ucByteValue ACCESS (ulADRString + CNr);
						ssByteValue := USINT_TO_INT(ucByteValue);

						IF bPair THEN
							ssChecksumm := ssChecksumm + ssByteValue;
							bPair := FALSE;
						ELSE
							ssChecksumm := ssChecksumm - ssByteValue;
							bPair := TRUE;
						END_IF
					END_FOR
				1:	(*character summ (9er) *)
					FOR CNr := 0 TO usUniStringLen DO
						ucByteValue ACCESS (ulADRString + CNr);
						ssByteValue := USINT_TO_INT(ucByteValue);

							ssChecksumm := ssChecksumm + ssByteValue;
					END_FOR
				ELSE
					ssChecksumm := 0;
					usChecksumm := 0;		(*prepared for later use*)
					usErrorCode := 12345;	(*THIS ChecksummMode IS NOT RELEASED NOW*)
			END_CASE
		END_IF
  		IF usErrorCode = 1 THEN usErrorCode := 0;  END_IF 	(*set state from BUSY to READY, if no errors occured*)

	END_IF

END_FUNCTION_BLOCK
```

#### UniXMLStri.typ - Exported data types
```iecst
(********************************************************************
 * COPYRIGHT -- INNIO Company
 ********************************************************************
 * Library: UniDecoXML
 * File: UniDecoXML.typ
 * Author: ZengereS
 * Created: November 02, 2010
 ********************************************************************
 * Data types of library UniDecoXML
 ********************************************************************)

TYPE
	tFoundSeparators_Type : 	STRUCT
		Code : STRING[1]; (*XML code for datapoint*)
		Length : UINT;
		Pos : UINT;
	END_STRUCT;
	tSeparators_Type : 	STRUCT
		Code : STRING[1]; (*XML code for datapoint*)
		VarName : STRING[32]; (*Variablename in TypeStructure (32characters signifikant)*)
		VarAdress : UDINT; (*Memory adress of variabe element in TypeStructure*)
		length : UDINT; (*size of variabe element in TypeStructure*)
		VarType : USINT; (*prepared for later use: variabe type of variabe element in TypeStructure*)
	END_STRUCT;
END_TYPE
```

#### UniXMLStri.var - Exported constants
```iecst
(********************************************************************
 * COPYRIGHT -- INNIO Company
 ********************************************************************
 * Library: UniDecoXML
 * File: UniDecoXML.var
 * Author: ZengereS
 * Created: November 02, 2010
 ********************************************************************
 * Constants of library UniDecoXML
 ********************************************************************)
VAR CONSTANT
	ERR_STATE : USINT := 252; (*Error State*)
END_VAR
```

#### UniXMLStri.fun - Exported functions and function blocks
```iecst
(********************************************************************
 * COPYRIGHT -- INNIO Company
 ********************************************************************
 * Library: UniXMLStri
 * File: UniDecoXML.fun
 * Author: ZengereS
 * Created: November 02, 2010
 ********************************************************************
 * Functions and function blocks of library UniXMLStri
 ********************************************************************)

FUNCTION_BLOCK xUniCodString
	VAR_INPUT
		bEnable : BOOL; (*TRUE = enable FUB*)
		ulXMLDataAdress : UDINT;
		ulXMLDataSize : UDINT;
	END_VAR
	VAR_OUTPUT
		bErrUniXMLRead : BOOL;
		usErrorCode : UINT; (*0=OK, ready*)
		bUniAnaFileReadDone : BOOL;
	END_VAR
	VAR
		bUniXMLWrite : BOOL;
		step : USINT; (*Internal step counter*)
	END_VAR
END_FUNCTION_BLOCK

FUNCTION_BLOCK xUniDecoString
	VAR_INPUT
		bEnable : BOOL; (*TRUE = enable FUB*)
		szConfigString : STRING[300];
		szSeparator : STRING[16]; (*Enter a combination of detectable separator characters here ( * = position will be ignored)*)
		ucStartPos : USINT; (*position of first character in string to start searching*)
	END_VAR
	VAR_OUTPUT
		usErrorCode : UINT; (*0=OK, ready*)
		usFoundPos : UINT; (*position of first data character after the found separator*)
		usFoundLenght : UINT; (*lenght of data in characters after the found separator*)
		bLastData : BOOL; (*TRUE, if no more separators will follow afther the found one*)
	END_VAR
	VAR
		CNr : UINT; (*Internal*)
		szCNr : STRING[1]; (*Internal*)
		usUniStringLen : UINT; (*Internal*)
		usUniSepaLen : UINT; (*Internal*)
		bFound : BOOL; (*Internal*)
		szWildcard : ARRAY[0..1] OF STRING[1]; (*Internal*)
		Sepa : UINT; (*Internal*)
		szSepar : ARRAY[0..16] OF STRING[1]; (*Internal*)
		ucFoundSlashs : USINT; (*Internal: count max number of following / characters*)
		ucFoundWildcards : USINT; (*Internal: count max. number of following wildcard characters*)
		CNrStartDetailSearch : UINT; (*internal*)
	END_VAR
END_FUNCTION_BLOCK

FUNCTION_BLOCK xUniCalcCheckSumm
	VAR_INPUT
		bEnable : BOOL; (*TRUE = enable FUB*)
		InString : STRING[300]; (*input string to calculate checksumm from*)
		usChecksummMode : USINT; (*0=alternating checksumm (dafeult), 1= prepared for later use...*)
		InMemAdress : UDINT; (*ALTERNATIVE INPUT to InString: enter memory adress in here to check*)
		InMemLenght : UINT; (*ALTERNATIVE INPUT to InString: enter memory lenght to check in combination with adress*)
	END_VAR
	VAR_OUTPUT
		ssChecksumm : INT; (*calculated checksumm from InString*)
		usChecksumm : UINT; (*calculated checksumm from InString without negative results*)
		usErrorCode : UINT; (*0=OK, ready*)
	END_VAR
	VAR
		CNr : UINT; (*Internal*)
		ulADRString : UDINT; (*internal*)
		usUniStringLen : UINT; (*internal*)
		bPair : BOOL; (*internal*)
		ucByteValue : REFERENCE TO USINT; (*internal*)
		ssByteValue : INT; (*internal*)
	END_VAR
END_FUNCTION_BLOCK
```

### Library Logical/Libraries/HALioBase (IEC, version 0.23.0)
Depends on: AsXml, AsIecCon, Runtime, sys_lib, asstring, DataObj

#### HALioBase.typ - Exported data types
```iecst
(********************************************************************
 * COPYRIGHT -- Bernecker + Rainer
 ********************************************************************
 * Library: HALioBase
 * File: HALioBase.typ
 * Author: froehlichw
 * Created: October 03, 2011
 ********************************************************************
 * Data types of library HALioBase
 *
 * History:
 * 03.01.2012  V0.00.0 froehlichw
 *      (new)  created
 * 07.03.2012  V0.10.0 froehlichw
 *   (change)  Qual to GoodQual
 *             in HALioAi_Type, HALioAi_INT_Type and HALioDi_Type
 * 30.07.2018  V0.13.1 Hohensinner
 *   (added)  Exist
 * 25.01.2023  V0.22.0 Perktold
 *    (change) Filter from INT to UINT in HALioExtern_Type
 * 31.01.2024  V0.23.0 Astner
 *    (change) Added Exist to DI,AO,DO; added GoodQual to AO,DO
 ********************************************************************)

TYPE
	HALioAi_Type : 	STRUCT
		Ai : REAL;
		Unfilt : REAL;
		GoodQual : BOOL;
		Exist : BOOL;
	END_STRUCT;
	HALioAi_INT_Type : 	STRUCT
		Ai : DINT;
		Unfilt : DINT;
		GoodQual : BOOL;
		Exist : BOOL;
	END_STRUCT;
	HALioDi_Type : 	STRUCT
		Di : BOOL;
		GoodQual : BOOL;
		Exist : BOOL;
	END_STRUCT;
	HALioAo_Type : 	STRUCT
		Ao : REAL;
		GoodQual : BOOL;
	END_STRUCT;
	HALioDo_Type : 	STRUCT
		Do : BOOL;
		GoodQual : BOOL;
	END_STRUCT;
	HALioExtern_Type : 	STRUCT
		Qual_Min : INT;
		Qual_Max : INT;
		Scal_X1 : DINT;
		Scal_X2 : DINT;
		Scal_Y1 : REAL;
		Scal_Y2 : REAL;
		Filter : UINT;
		HW_Type : USINT;
	END_STRUCT;
	HALioReaderPara_Type : 	STRUCT
		nodeName : STRING[99];
		nodeValue : STRING[99];
		nodeType : UDINT;
		nodeDepth : UDINT;
		attributeCount : UDINT;
		attributeIndex : UDINT;
		attributeMax : UDINT;
		attribute : ARRAY[0..3]OF HALioXmlAttribute_Type;
		checkType : HALioCheckType_Enum;
		checkPar : HALioCheckPar_Enum;
		pvAppName : STRING[39];
		pvName : STRING[39];
		pvAdr : UDINT;
		pvLen : UDINT;
		actIoChannel : UINT;
		pvParChecked : UINT;
		empty : BOOL;
		versionChecked : BOOL;
		pvChecked : BOOL;
		pvAllParChecked : BOOL;
	END_STRUCT;
	HALioXmlAttribute_Type : 	STRUCT
		name : STRING[99];
		value : STRING[99];
	END_STRUCT;
	HALioFubStep_Enum :
		(
		halSTP_INIT := 0, (* init FUB *)
		halSTP_GET_CONFIG := 5, (* get config module *)
		halSTP_CREATE_READER := 10, (* create XML reader *)
		halSTP_READ_NODE := 20, (* read XML node *)
		halSTP_READ_ATTRIBUTE := 25, (* read XML attribute *)
		halSTP_CHECK_DATA := 30, (* check data *)
		halSTP_ERROR := 90, (* error *)
		halSTP_CLOSE_READER := 99, (* close reader *)
		halSTP_FINISHED := 100 (* finished *)
		);
	HALioCheckType_Enum :
		(
		halCHK_VERSION := 0,
		halCHK_PV_NAME,
		halCHK_PV_PAR,
		halCHK_NOTHING := 99
		);
	HALioCheckPar_Enum :
		(
		halCHK_PAR_ACTIVE := 0,
		halCHK_PAR_TYPE,
		halCHK_PAR_QUAL_MIN,
		halCHK_PAR_QUAL_MAX,
		halCHK_PAR_MSG_NUM,
		halCHK_PAR_SCAL_X1,
		halCHK_PAR_SCAL_X2,
		halCHK_PAR_SCAL_Y1,
		halCHK_PAR_SCAL_Y2,
		halCHK_PAR_FILTER,
		halCHK_PAR_NOTHING := 99
		);
END_TYPE
```

#### HALioBase.var - Exported constants
```iecst
(********************************************************************
 * COPYRIGHT -- Bernecker + Rainer
 ********************************************************************
 * Library: HALioBase
 * File: HALioBase.var
 * Author: froehlichw
 * Created: October 03, 2011
 ********************************************************************
 * Constants of library HALioBase
 *
 * History:
 * 05.01.2012  V0.00.0 froehlichw
 *      (new)  created
 * 17.10.2012  V0.12.0 froehlichw
 *      (add)  Error numbers:
 *               halERR_SIGPV_LENGTH_NOT_MATCHING
 *               halERR_PARPV_LENGTH_NOT_MATCHING
 ********************************************************************)
(* Signal types digital in *)
VAR CONSTANT
	DI_NORMAL : UINT := 10;
	DI_NORMAL_INV : UINT := 11;
	DI_NORMAL_UR20 : UINT := 12;
	DI_NORMAL_INV_UR20 : UINT := 13;
END_VAR
(* Signal types digital out *)
VAR CONSTANT
	DO_NORMAL : UINT := 20;
	DO_NORMAL_UR20 : UINT := 21;
END_VAR
(* Signal types analog in *)
VAR CONSTANT
	AI_0_20mA_INT16 : UINT := 30;
	AI_0_10V_INT16 : UINT := 31;
	AI_10_10V_INT16 : UINT := 32;
	AI_TEMP_1_10C : UINT := 33;
	AI_INT8 : UINT := 34;
	AI_INT16 : UINT := 35;
	AI_INT32 : UINT := 36;
	AI_0_20mA_INT16_UR20 : UINT := 37;
	AI_0_10V_INT16_UR20 : UINT := 38;
	AI_10_10V_INT16_UR20 : UINT := 39;
	AI_TEMP_1_10C_UR20 : UINT := 40;
	AI_INT8_UR20 : UINT := 41;
	AI_INT16_UR20 : UINT := 42;
	AI_INT32_UR20 : UINT := 43;
END_VAR
(* Signal types analog out *)
VAR CONSTANT
	AO_0_20mA_INT16 : UINT := 50;
	AO_0_10V_INT16 : UINT := 51;
	AO_10_10V_INT16 : UINT := 52;
	AO_0_20mA_INT16_UR20 : UINT := 53;
	AO_0_10V_INT16_UR20 : UINT := 54;
	AO_10_10V_INT16_UR20 : UINT := 55;
END_VAR
(* Error numbers *)
VAR CONSTANT
	halERR_NO_ERROR : UINT := 0; (* no error *)
	halERR_SIGNAL_TYPE_UNKNOWN : UINT := 50000; (* unknown signal type *)
	halERR_INP_pSIGNAL_NV : UINT := 50001; (* pointer pSignal not valid *)
	halERR_INP_pPV_NAME_NV : UINT := 50002; (* pointer pPV_Name not valid *)
	halERR_INP_QUAL_MIN_EQ_MAX_NE_0 : UINT := 50003; (* input Qual_Min = Qual_Max but not 0*)
	halERR_INP_QUAL_MIN_GT_MAX : UINT := 50004; (* input Qual_Min > Qual_Max *)
	halERR_INP_pHALIOSIGNAL_NV : UINT := 50005; (* input pHALioSignal not valid or MaxNumIoChannels = 0 *)
	halERR_INP_SCAL_X1_EQ_X2_NE_0 : UINT := 50006; (* input Scal_X1 = Scal_X2 but not 0 *)
	halERR_INP_SCAL_Y1_EQ_Y2_NE_0 : UINT := 50007; (* input Scal_Y1 = Scal_Y2 but not 0 *)
	halERR_INP_FILTER_EQ_0 : UINT := 50008; (* input Filter = 0 *)
	halERR_CFG_MODULE_NOT_FOUND : UINT := 50020; (* configuration modul not found *)
	halERR_XML_READER : UINT := 50021; (* error with XML reader *)
	halERR_TOO_MANY_ATTRIBUTES : UINT := 50022; (* too many attributes defined *)
	halERR_READ_NODE : UINT := 50023; (* error reading node *)
	halERR_READ_ATTRIBUTE : UINT := 50024; (* error rerading attribute *)
	halERR_VERSION_NV : UINT := 50025; (* version of config module not valid *)
	halERR_PV_NOT_FOUND : UINT := 50026; (* PV not found *)
	halERR_PV_NAME_TOO_LONG : UINT := 50027; (* PV name too long *)
	halERR_PARAMETER_VALUE_NV : UINT := 50028; (* parameter value not valid *)
	halERR_PARAMETER_MISSING : UINT := 50029; (* parameter missing *)
	halERR_MAX_NUM_IOS_TOO_LOW : UINT := 50030; (* max number of IO Channels lower then needed *)
	halERR_SIGPV_LENGTH_NOT_MATCHING : UINT := 50031; (* signal PV lenght does not match to defined signal type *)
	halERR_PARPV_LENGTH_NOT_MATCHING : UINT := 50032; (* external parameter PV lenght of does not match *)
	halERR_FUB_NOT_ENABLED : UINT := 65534; (* FUB not enabled *)
	halERR_FUB_BUSY : UINT := 65535; (* FUB busy *)
END_VAR
(* node names *)
VAR CONSTANT
	halNODE_ROOT : STRING[20] := 'HALioConfiguration'; (* root node name *)
	halNODE_GROUP : STRING[20] := 'Group'; (* group node name *)
	halNODE_PARAMETER : STRING[20] := 'Parameter'; (* parameter node name *)
END_VAR
(* attribute names *)
VAR CONSTANT
	halATTR_VERSION : STRING[20] := 'Version'; (* attribute name Version *)
	halATTR_VERSION_VAL_1_0_00 : STRING[20] := '1.0.00'; (* attribute value Version 1.0.00 *)
	halATTR_PV_NAME : STRING[20] := 'PV_Name'; (* attribute name PV_Name *)
	halATTR_ID : STRING[20] := 'ID'; (* attribute name ID *)
	halATTR_VALUE : STRING[20] := 'Value'; (* attribute name Value *)
END_VAR
(* attribute ID values *)
VAR CONSTANT
	halATTR_ID_ACTIVE : STRING[20] := 'Active'; (* attribute ID value Active *)
	halATTR_ID_TYPE : STRING[20] := 'Type'; (* attribute ID value Type *)
	halATTR_ID_QUAL_MIN : STRING[20] := 'Qual_Min'; (* attribute ID value Qual_Min *)
	halATTR_ID_QUAL_MAX : STRING[20] := 'Qual_Max'; (* attribute ID value Qual_Max *)
	halATTR_ID_MSG_NUM : STRING[20] := 'Msg_Num'; (* attribute ID value Msg_Num *)
	halATTR_ID_SCAL_X1 : STRING[20] := 'Scal_X1'; (* attribute ID value Scal_X1 *)
	halATTR_ID_SCAL_X2 : STRING[20] := 'Scal_X2'; (* attribute ID value Scal_X2 *)
	halATTR_ID_SCAL_Y1 : STRING[20] := 'Scal_Y1'; (* attribute ID value Scal_Y1 *)
	halATTR_ID_SCAL_Y2 : STRING[20] := 'Scal_Y2'; (* attribute ID value Scal_Y2 *)
	halATTR_ID_FILTER : STRING[20] := 'Filter'; (* attribute ID value Filter *)
END_VAR
(* bit numbers of checked parameters *)
VAR CONSTANT
	halPAR_ACTIVE : UINT := 0; (* bit number 0 in pvParChecked *)
	halPAR_TYPE : UINT := 1; (* bit number 1 in pvParChecked *)
	halPAR_QUAL_MIN : UINT := 2; (* bit number 2 in pvParChecked *)
	halPAR_QUAL_MAX : UINT := 3; (* bit number 3 in pvParChecked *)
	halPAR_MSG_NUM : UINT := 4; (* bit number 4 in pvParChecked *)
	halPAR_SCAL_X1 : UINT := 5; (* bit number 5 in pvParChecked *)
	halPAR_SCAL_X2 : UINT := 6; (* bit number 6 in pvParChecked *)
	halPAR_SCAL_Y1 : UINT := 7; (* bit number 7 in pvParChecked *)
	halPAR_SCAL_Y2 : UINT := 8; (* bit number 8 in pvParChecked *)
	halPAR_FILTER : UINT := 9; (* bit number 9 in pvParChecked *)
END_VAR
```

#### HALioBase.fun - Exported functions and function blocks
```iecst
(********************************************************************
 * COPYRIGHT -- Bernecker + Rainer
 ********************************************************************
 * Library: HALioBase
 * File: HALioBase.fun
 * Author: froehlichw
 * Created: October 03, 2011
 ********************************************************************
 * Functions and function blocks of library HALioBase
 *
 * History:
 * 05.01.2012  V0.00.0 froehlichw
 *      (new)  created
 * 02.02.2022  V0.21.0 Schmid
 *    (added)  Reset
 *             in HALioFilter, HALioFilterR
 * 25.01.2023  V0.22.0 Perktold
 *    (added)  TaskClass and CycleTimeMs in HALioSignal
 *    (change) Filter from UINT to REAL in HALioFilterR
 *    (added)  evalHALioSignal
 ********************************************************************)

FUNCTION_BLOCK HALioCfg (* configurates inputs of HALioSignal *)
	VAR_INPUT
		enable : BOOL;
		pCfgModDevice : UDINT;
		pCfgModName : UDINT;
		pAppModName : UDINT;
		pHALioSignal : UDINT;
		MaxNumIoChannels : UINT;
	END_VAR
	VAR_OUTPUT
		ParOK : BOOL;
		ActNumIoChannels : UINT;
		CfgModError : BOOL;
		pErrInfo1 : UDINT;
		pErrInfo2 : UDINT;
		pErrInfo3 : UDINT;
		status : UINT;
	END_VAR
	VAR
		stepFub : HALioFubStep_Enum;
		para : HALioReaderPara_Type;
		HALioSignal_0 : REFERENCE TO HALioSignal;
		DatObjInfo_0 : DatObjInfo;
		xmlCreateMemoryReader_0 : xmlCreateMemoryReader;
		xmlReadNextNode_0 : xmlReadNextNode;
		xmlReadAttributeNr_0 : xmlReadAttributeNr;
		xmlCloseMemoryReader_0 : xmlCloseMemoryReader;
		nextAdr : UDINT;
		pEmptyString : UDINT;
		pvName : STRING[99];
		strErrNb : STRING[15];
		status_PV_xgetadr : UINT;
		strLen : UINT;
		strLenMax : UINT;
		Type : UINT;
		iVal : DINT;
		rVal : REAL;
		pVal : REFERENCE TO USINT;
		sigAi : HALioAi_Type;
		sigAi_INT : HALioAi_INT_Type;
		sigAo : HALioAo_Type;
		sigDi : HALioDi_Type;
		sigDo : HALioDo_Type;
		sigExtPar : HALioExtern_Type;
		zzEdge00000 : BOOL;
	END_VAR
END_FUNCTION_BLOCK

FUNCTION_BLOCK HALioSignal (* signal processing *)
	VAR_INPUT
		ParOK : BOOL;
		HwOK : BOOL;
		Active : BOOL;
		Type : UINT;
		Qual_Min : INT;
		Qual_Max : INT;
		Scal_X1 : DINT;
		Scal_X2 : DINT;
		Scal_Y1 : REAL;
		Scal_Y2 : REAL;
		Filter : UINT;
		pExtern : UDINT;
		pPV_Name : UDINT;
		pMsg : UDINT;
		pSignal : UDINT;
		TaskClass : UDINT;
		CycleTimeMs : REAL;
	END_VAR
	VAR_OUTPUT
		status : UINT;
	END_VAR
	VAR
		sigAi : REFERENCE TO HALioAi_Type;
		sigAi_INT : REFERENCE TO HALioAi_INT_Type;
		sigAo : REFERENCE TO HALioAo_Type;
		sigDi : REFERENCE TO HALioDi_Type;
		sigDo : REFERENCE TO HALioDo_Type;
		ain : REFERENCE TO INT;
		ain_INT8 : REFERENCE TO SINT;
		ain_INT16 : REFERENCE TO INT;
		ain_INT32 : REFERENCE TO DINT;
		ainVal : DINT;
		aout : REFERENCE TO INT;
		din : REFERENCE TO BOOL;
		dout : REFERENCE TO BOOL;
		msg : REFERENCE TO BOOL;
		isInput : BOOL;
		isOutput : BOOL;
		aiMinMax : BOOL;
		extPar : REFERENCE TO HALioExtern_Type;
		parUse : HALioExtern_Type;
		HALioFilter_0 : HALioFilter;
		HALioFilterR_0 : HALioFilterR;
	END_VAR
END_FUNCTION_BLOCK

FUNCTION_BLOCK HALioFilter (* filter with PT1 behaivior and DINT in/output *)
	VAR_INPUT
		In : DINT;
		Filter : UINT;
		Reset : BOOL;
	END_VAR
	VAR_OUTPUT
		Out : DINT;
	END_VAR
	VAR
		mw : DINT;
	END_VAR
END_FUNCTION_BLOCK

FUNCTION_BLOCK HALioFilterR (* filter with PT1 behaivior and REAL in/output *)
	VAR_INPUT
		In : REAL;
		Filter : REAL;
		Reset : BOOL;
	END_VAR
	VAR_OUTPUT
		Out : REAL;
	END_VAR
	VAR
		mw : LREAL;
	END_VAR
END_FUNCTION_BLOCK

FUNCTION HALioSigscal : DINT (* signal scaling In DINT / Out DINT *)
	VAR_INPUT
		In : DINT;
		X1 : DINT;
		X2 : DINT;
		Y1 : DINT;
		Y2 : DINT;
	END_VAR
END_FUNCTION

FUNCTION HALioSigscalR : REAL (* signal scaling In DINT / Out REAL *)
	VAR_INPUT
		In : DINT;
		X1 : DINT;
		X2 : DINT;
		Y1 : REAL;
		Y2 : REAL;
	END_VAR
END_FUNCTION

FUNCTION HALioSigscalRInv : DINT (* signal scaling In REAL / Out DINT *)
	VAR_INPUT
		In : REAL;
		X1 : REAL;
		X2 : REAL;
		Y1 : DINT;
		Y2 : DINT;
	END_VAR
END_FUNCTION

FUNCTION evalHALioSignal : UINT (*evaluate IO signal*)
	VAR_INPUT
		ParOK : BOOL;
		HwOK : BOOL;
		ActNumIoChannels : UINT;
		CycleTimeMs : REAL;
	END_VAR
	VAR_IN_OUT
		xHALioSignal : ARRAY[0..1299] OF HALioSignal;
		SignalError : UINT;
		SignalErrorIdx : UINT;
	END_VAR
	VAR
		idx : UINT;
	END_VAR
END_FUNCTION
```
